{attribute 'GeneratedUsingTerminal: EL3024-0000-0019'}
{attribute addProperty BoxType "EL3024-0000-0019"}
{attribute addProperty Id "WcStateAT %I*BOOL1InputToggleAT %I*BOOL1"}
{attribute addProperty CRC "2425479403"}
{attribute addProperty Size "2"}
TYPE WcState_9091E0EB EXTENDS WcStateInputToggleBase_F68C23A9 :
STRUCT
	{attribute addProperty Name "WcState"}
	WcState AT %I* : BOOL;
	{attribute addProperty Name "InputToggle"}
	InputToggle AT %I* : BOOL;
END_STRUCT
END_TYPE

(* stored: Version 1.2.0.0, ProductVersion 3.1.4024.9
   DUT WcState_9091E0EB: Id {51ba3f53-c7b6-4eaf-b63f-14b791611ee4} *)
